// TIA Portal V16 export
// export: Created 2024-09-05T17:39:24.4956809Z, ExportSetting WithDefaults, DisplayName Totally Integrated Automation Portal, DisplayVersion V16 Update 6, DisplayName TIA Portal Version Control Interface, DisplayVersion V16 Update 2, DisplayName TIA Portal Openness, DisplayVersion V16 Update 6, DisplayName STEP 7 Professional, DisplayVersion V16 Update 6, DisplayName STEP 7 Safety, DisplayVersion V16, DisplayName WinCC Advanced, DisplayVersion V16 Update 6
FUNCTION "Extract_data_DMC" : Void   // FC2011, LAD
{ S7_Optimized_Access := 'TRUE' }
VERSION : 0.1
// stored: AutoNumber false, IsIECCheckEnabled false, SetENOAutomatically false, UDAEnableTagReadback false
   VAR_INPUT
      round : Byte;
      Data_DMC : Array[1.."MaxRoundNumber", 1..10] of "DATA_DMC";
   END_VAR
   VAR_OUTPUT
      DATA_DMC_Extract : Array[1..10] of String[25];
   END_VAR
   VAR_TEMP
      idx : SInt;
      round_idx : SInt;
   END_VAR
BEGIN

REGION Network 1
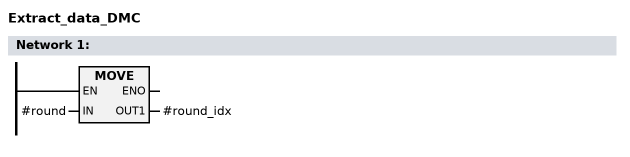
   RUNG wire#powerrail
      Move(in := #round, out1 => #round_idx)
   END_RUNG
   // the same network as SCL:
   #round_idx := #round;
END_REGION

REGION Network 2 (SCL)
   FOR #idx := 1 TO 10 DO
       #DATA_DMC_Extract[#idx] := #Data_DMC[#round_idx, #idx].SAP_REF_PRODUCTION;

   END_FOR;
END_REGION
END_FUNCTION
